FUNCTION_BLOCK TExampleInterfaceImplementation IMPLEMENTS IExampleInterface
VAR_INPUT
END_VAR
VAR_OUTPUT
END_VAR
VAR
END_VAR

END_FUNCTION_BLOCK

(* stored: Version 1.1.0.1, ProductVersion 3.1.4024.3
   POU TExampleInterfaceImplementation: Id {f249db92-7f44-46a0-b7fe-a467b8ef1444}, SpecialFunc None *)
